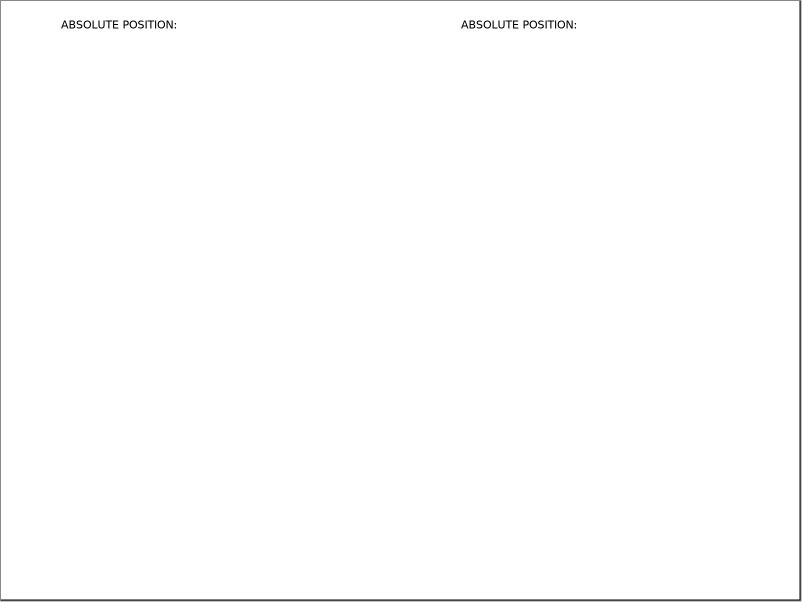
VISUALIZATION F06_Read_Bool_Parameter  // 802x602
    Rectangle (0,0 800x600)
    Label (10,10 170x30), "ABSOLUTE POSITION:"
    Label (410,10 170x30), "ABSOLUTE POSITION:"
END_VISUALIZATION

(* stored: Version 1.1.0.1, ProductVersion 3.1.4022.7
   Visu F06_Read_Bool_Parameter: Id {6aefa094-05b2-407e-b962-e656772ee619} *)
